// TIA Portal project "node_RED1" (V14)

(* hardware
DEVICE "S7-1200 station_1"  S7-1200 Station
   slot 0: "Rack_0"  S7-1200 Rack  Rack  V1.0
   slot 1: "PLC_1"  CPU 1214C DC/DC/DC  6ES7 214-1AG40-0XB0  V4.2
   slot 3: "AQ 1x12BIT_1"  AQ1 signal board  6ES7 232-4HA30-0XB0  V1.0
*)

// ===== PLC "PLC_1"  CPU 1214C DC/DC/DC =====

VAR_GLOBAL   // PLC tag table "Default tag table"
   "Clock_Byte" AT %MB0 : Byte;
   "Clock_10Hz" AT %M0.0 : Bool;
   "Clock_5Hz" AT %M0.1 : Bool;
   "Clock_2.5Hz" AT %M0.2 : Bool;
   "Clock_2Hz" AT %M0.3 : Bool;
   "Clock_1.25Hz" AT %M0.4 : Bool;
   "Clock_1Hz" AT %M0.5 : Bool;
   "Clock_0.625Hz" AT %M0.6 : Bool;
   "Clock_0.5Hz" AT %M0.7 : Bool;
   "analogni vhod" AT %IW64 : Word;
   "analogniIZHOD" AT %QW80 : Word;
   "digitalniVHODI" AT %IW0 : Word;
   "digitalniIZHODI" AT %QW0 : Word;
   "pomnilnik0" AT %MW400 : Int;
END_VAR

DATA_BLOCK "globalne"   // DB1
{ S7_Optimized_Access := 'FALSE' }
VERSION : 0.1
   VAR
      stikala : Word;
      target : UInt := 2000;
      analogni : UInt;
      digitalniIzhodi : Word;
      stevec : Int := 77;
      analogni_izhod : UInt;
      niz_1 : String;
      vpis : Int;
      nova : Bool;
      niz : Array[0..20] of Byte;
      stara : Bool;
      test : Word;
   END_VAR
BEGIN
END_DATA_BLOCK

DATA_BLOCK "vpisujem"   // DB2
{ S7_Optimized_Access := 'FALSE' }
VERSION : 0.1
   VAR
      vpis : Int;
   END_VAR
BEGIN
END_DATA_BLOCK

DATA_BLOCK "nizi123"   // DB3
{ S7_Optimized_Access := 'FALSE' }
VERSION : 0.1
   VAR
      niz3 : String;
   END_VAR
BEGIN
END_DATA_BLOCK

DATA_BLOCK "branje"   // DB4
{ S7_Optimized_Access := 'FALSE' }
VERSION : 0.1
   VAR
      vlaga : Int;
   END_VAR
BEGIN
END_DATA_BLOCK

ORGANIZATION_BLOCK "Main"   // OB1, SCL, ProgramCycle
TITLE = "Main Program Sweep (Cycle)"
{ S7_Optimized_Access := 'TRUE' }
VERSION : 0.1
   VAR_INPUT
      Initial_Call : Bool;   // Initial call of this OB
      Remanence : Bool;   // =True, if remanent data are available
   END_VAR
   VAR_TEMP
      steje : Bool;
      string1 : String;
      i : Int;
      digitalniVhodiNiz : String;
      digitalniIzhodiNiz : String;
      nizanalog : String;
      mojArray : Array[0..24] of Byte;
   END_VAR
BEGIN
   // Datum: 18. januar 2020 -- povezava preko node-red na spletno stran

   "globalne".analogni := WORD_TO_UINT("analogni vhod");
   "analogniIZHOD":="globalne".analogni_izhod;


   //"digitalniIZHODI" := 16#3333;
   "globalne".stikala :=  "digitalniVHODI";
   "digitalniIZHODI":=UINT_TO_WORD("globalne".digitalniIzhodi);
   #digitalniVhodiNiz := S_CONV((WORD_TO_UINT("digitalniVHODI")));
   #digitalniIzhodiNiz := S_CONV((WORD_TO_UINT("digitalniIZHODI")));
   #nizanalog := S_CONV("globalne".analogni);
   "globalne".niz_1 := #nizanalog;
   "globalne".niz_1 := CONCAT(IN1:= "globalne".niz_1, IN2:= '#');
   "globalne".niz_1 := CONCAT(IN1 := "globalne".niz_1, IN2 := #digitalniVhodiNiz);
   "globalne".niz_1 := CONCAT(IN1 := "globalne".niz_1, IN2 := '#');
   "globalne".niz_1 := CONCAT(IN1 := "globalne".niz_1, IN2 :=#digitalniIzhodiNiz);





   IF "globalne".stevec > 2000 THEN
       "globalne".stevec := 0;
   END_IF;
   "branje".vlaga := "globalne".stevec;




   #string1:='Lep pozdrav PLC!';
   "nizi123".niz3 := 'Lep pozdrav!';

   "globalne".nova := "Clock_1Hz";
   #steje := "globalne".stara AND NOT "globalne".nova;
   IF #steje=TRUE THEN
       "globalne".stevec:="globalne".stevec+1;
   END_IF;
   "globalne".stara := "globalne".nova;

   "pomnilnik0" := "globalne".stevec;


   IF ("globalne".target > "globalne".analogni) THEN
       "digitalniIZHODI" := 16#ffff;
   ELSE
       "digitalniIZHODI" := 0;
   END_IF;
END_ORGANIZATION_BLOCK